FUNCTION_BLOCK FB_Tracking
VAR_IN_OUT
	stAxis  : ARRAY [GVL.cXP .. GVL.cXM] OF ST_AxisGroup;	
END_VAR
VAR_INPUT
	eCommand 			: E_Commands;
	bMotionDone			: BOOL;
	inReset				: ST_Reset;
	inMoveAxisAbsolute	: ST_MoveAxisAbsolute;
	inMoveAxisRelative	: ST_MoveAxisRelative;
END_VAR
VAR_OUTPUT
	stOutMotionDone : ST_MotionDone;
END_VAR
VAR
	//used in tracking Action
	stTrack			: ARRAY [0 .. 4] OF ST_TRACK;
	stTrackTemp		: ST_TRACK;
	bGoNextSeq		: BOOL;
	nAxisID			: INT;
	tTimeEnd		: T_DCTIME64;
	nMask			: ULINT := 16#FFFF_FFFF_0000_0000;
	
	//used in determining target duration
	fSpeed			: LREAL;
	tTargetDur		: LTIME;
	fDistance		: LREAL;
	
	fbMoving_Rtrig : ARRAY[0 .. 1] OF R_TRIG;
	fbRtrig		: ARRAY[GVL.cHallLower..GVL.cHallUpper] OF R_Trig;
	bInMotion	: BOOL;
	stMotionDone : ARRAY [0..1] OF ST_MotionDone;	
	nSequence	: DINT;
	nLastMoved	: INT;
	
	//counter
	i, j, k, m		: INT := 0;
	nTPC	: INT; //Trip Per Cycle
	
	//TestVar
	testRtrig : R_TRIG;
	testRtrig2 : R_TRIG;
	testInt: INT;
	testInt2: INT;
	testInt3: INT;
	testInt4: INT;
	testInt5: INT;
	testInt6: INT;
	testLREAL : LREAL;
	testTemp : ARRAY[0 .. 4] OF ST_Track;
	testTime : ARRAY[0 .. 4] OF T_DCTIME64;
	teststTrack : ARRAY[0 .. 4] OF T_DCTIME64;
	testDCTime	: ARRAY[0 .. 4] OF T_DCTIME64;
	nMask2	 : ULINT := 16#0000_0000_FFFF_FFFF;
	a, b : INT;
	
	
	
END_VAR

//////////////////////////////////////////////////////////////
//Algorithm for tracking blade position using hall switches	//
//////////////////////////////////////////////////////////////
stAxis[GVL.cXP].bTrackedFlag:=FALSE;
stAxis[GVL.cXM].bTrackedFlag:=FALSE;
nTPC:=0;
testInt3:=0;
testInt4:=0;

fbMoving_Rtrig[GVL.cXP](CLK:=stAxis[GVL.cXP].axisRef.Status.Moving);
IF fbMoving_Rtrig[GVL.cXP].Q THEN
	bInMotion:=TRUE;
	//AxisXP
	stMotionDone[GVL.cXP].axisNum := GVL.cXP;
	stMotionDone[GVL.cXP].nsamples := 0;
	stMotionDone[GVL.cXP].ntrans := 0;
	stMotionDone[gvl.cXP].startPos := stAxis[GVL.cXP].axisRef.NcToPlc.ActPos;
	stMotionDone[GVL.cXP].startTime := F_GetCurDcTaskTime64();
	stMotionDone[GVL.cXP].targetDur := LTIME#0D0H0M0S0MS0US0NS;
END_IF
fbMoving_Rtrig[GVL.cXM](CLK:=stAxis[GVL.cXM].axisRef.Status.Moving);
IF fbMoving_Rtrig[GVL.cXM].Q THEN
	bInMotion:=TRUE;
	//AxisXM
	stMotionDone[gvl.cXM].axisNum := GVL.cXM;
	stMotionDone[gvl.cXM].nsamples := 0;
	stMotionDone[gvl.cXM].ntrans := 0;
	stMotionDone[gvl.cXM].startPos := stAxis[GVL.cXM].axisRef.NcToPlc.ActPos;
	stMotionDone[gvl.cXM].startTime := F_GetCurDcTaskTime64();
	stMotionDone[gvl.cXM].targetDur := LTIME#0D0H0M0S0MS0US0NS;
END_IF

//determine target duration
IF eCommand = E_Commands.takeExposure THEN
	fSpeed	:= inReset.speed;
	IF (fSpeed>0) THEN
		IF (fSpeed>1668.355556) THEN
			fSpeed:=1668.355556;
		END_IF
		tTargetDur 	:= LREAL_TO_LTIME((2*GVL.cPosEnd)/(fSpeed)*EXPT(10,9));
	END_IF
ELSIF eCommand = E_Commands.moveAxisAbsolute THEN
	fDistance := ABS(stAxis[inMoveAxisAbsolute.axisIndex].axisRef.NcToPlc.ActPos - inMoveAxisAbsolute.position);
	fSpeed	:= inMoveAxisAbsolute.speed;
	IF (fSpeed>0) THEN
		IF (fSpeed>1668.355556) THEN
			fSpeed:=1668.355556;
		END_IF
		tTargetDur 	:= LREAL_TO_LTIME(((2*fDistance)/(fSpeed))*EXPT(10,9));
	END_IF
ELSIF eCommand = E_Commands.moveAxisRelative THEN
	tTargetDur	:= TIME_TO_LTIME(inMoveAxisRelative.moveTime);
END_IF

//Checks to see which blade set last moved
IF (stAxis[GVL.cXM].axisRef.Status.Moving AND stAxis[GVL.cXP].axisRef.Status.InTargetPosition) THEN
	nLastMoved:=GVL.cXM;
ELSIF (stAxis[GVL.cXP].axisRef.Status.Moving AND stAxis[GVL.cXM].axisRef.Status.InTargetPosition) THEN
	nLastMoved:=GVL.cXP;
END_IF
IF bMotionDone THEN
	//use for determining which blade set has finished during a travelling slit motion
	IF (stAxis[GVL.cXM].axisRef.Status.Moving AND stAxis[GVL.cXP].axisRef.Status.InTargetPosition) THEN
		nAxisID:=GVL.cXP;
	ELSIF (stAxis[GVL.cXP].axisRef.Status.Moving AND stAxis[GVL.cXM].axisRef.Status.InTargetPosition) THEN
		nAxisID:=GVL.cXM;
	ELSE 
		nAxisID:=nLastMoved;
	END_IF
	//bInMotion flag remains true if any of the blade set is still in motion
	IF ((NOT stAxis[GVL.cXP].axisRef.Status.Moving) AND (NOT stAxis[GVL.cXM].axisRef.Status.Moving)) THEN
		bInMotion := FALSE;
	END_IF
	nSequence := nSequence+1;
	tTimeEnd := F_GetCurDcTaskTime64();
	stMotionDone[nAxisID].actualDur := ULINT_TO_LTIME(tTimeEnd-stMotionDone[nAxisID].startTime);
	stMotionDone[nAxisID].targetDur := tTargetDur;
	stMotionDone[nAxisID].targetPos := stAxis[nAxisID].axisRef.NcToPlc.TargetPos;
	stMotionDone[nAxisID].endPos := stAxis[nAxisID].axisRef.NcToPlc.ActPos;
	
	stOutMotionDone:=stMotionDone[nAxisID];
	stOutMotionDone.sequence:=nSequence;
END_IF


//Detect hall switch transitions
FOR i:=GVL.cHallLower TO GVL.cHallUpper BY 1 DO
	fbRtrig[i](CLK:=GVL.nNumOfInputs[i].0);
	IF fbRtrig[i].Q THEN
		//identifies which hall switch tripped
		stTrack[nTPC].nSeqToCompare := INT_TO_WORD((i*10)+5);
		stTrack[nTPC].bEdgeToCompare := GVL.bInputEventState[i];
		stTrack[nTPC].nHallID := i;
		(*
			The time-stamping module only keeps track of the lower 32-bit time (about 4.29 seconds).
			To get the actual 64-bit time, add the acquired 32-bit time to the upper 32 bit of the DC time. 
			Check to see if the event time has overflowed by comparing appended time with current DC task time. 
			If appeneded time is greater than dc task time, then the 32-bit clock has overflowed.
			Decrement the 33rd bit of the appended time by 1 to get the correct time.
		*)
		stTrack[nTPC].tScanTime := (F_GetCurDcTaskTime64() AND nMask) + GVL.nInputEventTime[stTrack[nTPC].nHallID];
		IF stTrack[nTPC].tScanTime > F_GetCurDcTaskTime64() THEN
			stTrack[nTPC].tScanTIME := stTrack[nTPC].tScanTime - 16#1_0000_0000;
			testInt5:=testInt5+1;
		END_IF
		//increment the index
		nTPC:=nTPC+1;
		
		//Sort the data from lowest time to highest time
		IF nTPC>=2 THEN
			FOR j:=nTPC-1 TO 1 BY -1 DO
				IF (stTrack[j].tScanTime < stTrack[j-1].tScanTime) THEN
						stTrackTemp := stTrack[j];
						stTrack[j] := stTrack[j-1];
						stTrack[j-1] := stTrackTemp;
						testInt6 := testInt6+1;
				END_IF
			END_FOR
		END_IF

		
		//For debugging only: To see the highest number of trip per cycle
		testRTrig2(CLK:=(nTPC>=2));
		IF testRTrig2.Q THEN
			testInt3 := 1;
		END_IF
		testRTrig(CLK:=(nTPC>=3));
		IF testRTrig.Q THEN
			testTemp := stTrack;
			testInt4 := 1;
		END_IF
		IF m<nTPC THEN
			m:= nTPC;
		END_IF
		

			IF ((F_GetCurDcTaskTime64() - stTrack[0].tScanTime)>2000000) AND nTPC=1 THEN
				testTime[0]	:= F_GetCurDcTaskTime64() - stTrack[0].tScanTime;
				teststTrack[0] := stTrack[0].tScanTime;
				 testDCTime[0] := F_GetCurDcTaskTime64();
			END_IF
			IF ((F_GetCurDcTaskTime64() - stTrack[1].tScanTime)>2000000) AND nTPC=2 THEN
				testTime[1]	:= F_GetCurDcTaskTime64() - stTrack[1].tScanTime;
				teststTrack[1] := stTrack[1].tScanTime;
				testDCTime[1] := F_GetCurDcTaskTime64();
			END_IF
			IF ((F_GetCurDcTaskTime64() - stTrack[2].tScanTime)>2000000) AND nTPC=3 THEN
				testTime[2]	:= F_GetCurDcTaskTime64() - stTrack[2].tScanTime;
				teststTrack[2] := stTrack[2].tScanTime;
				testDCTime[2] := F_GetCurDcTaskTime64();
			END_IF
			IF ((F_GetCurDcTaskTime64() - stTrack[3].tScanTime)>2000000) AND nTPC=4 THEN
				testTime[3]	:= F_GetCurDcTaskTime64() - stTrack[3].tScanTime;
				teststTrack[3] := stTrack[3].tScanTime;
				testDCTime[3] := F_GetCurDcTaskTime64();
			END_IF
	END_IF
	
	//For debugging - checks to see if the same hall switch is tripped twice in one cycle
	IF GVL.nNumOfInputs[i]=2 THEN
		testInt:=testint+1;
	END_IF
	
END_FOR


	
//blade motion tracking
IF nTPC>0 THEN
	FOR k:=0 TO nTPC-1 BY 1 DO
		IF (stAxis[GVL.cXP].axisRef.Status.Moving AND stAxis[GVL.cXM].axisRef.Status.Moving) AND
			(stAxis[GVL.cXP].axisRef.Status.PositiveDirection AND stAxis[GVL.cXM].axisRef.Status.PositiveDirection) THEN
			ACT_TrackingDoublePositive();
		ELSIF (stAxis[GVL.cXP].axisRef.Status.Moving AND stAxis[GVL.cXM].axisRef.Status.Moving) AND
			(stAxis[GVL.cXP].axisRef.Status.NegativeDirection AND stAxis[GVL.cXM].axisRef.Status.NegativeDirection) THEN
			ACT_TrackingDoubleNegative();
		ELSE
			ACT_TrackingSingle();
		END_IF
		bGoNextSeq:=FALSE;
		IF nTPC=2 THEN
			testInt2:=testInt2+1;
		END_IF
	END_FOR
END_IF

ACTION ACT_TrackingDoubleNegative:
//Hall sensors position tracking for axis XP
IF stAxis[GVL.cXP].axisRef.Status.Moving THEN
	//Compare current sequence with recorded sequence. Update position if match. Negative direction.
	IF stAxis[GVL.cXP].axisRef.status.NegativeDirection AND stAxis[GVL.cXP].stHall[GVL.cDirNeg, stAxis[GVL.cXP].nTripCount].nSeq = stTrack[k].nSeqToCompare AND
			stAxis[GVL.cXP].stHall[GVL.cDirNeg, stAxis[GVL.cXP].nTripCount].bEdge = stTrack[k].bEdgeToCompare AND (NOT bGoNextSeq) THEN
		stAxis[GVL.cXP].fHallPosAct := stAxis[GVL.cXP].fHallPosCal[GVL.cDirNeg, stAxis[GVL.cXP].nTripCount];
		stAxis[GVL.cXP].nTripCount := stAxis[GVL.cXP].nTripCount - 1;		
		//track difference between hall sensor and encoder data at trip point
		stAxis[GVL.cXP].fPosDiffAtTrip := stAxis[GVL.cXP].axisRef.NcToPlc.ActPos - stAxis[GVL.cXP].fHallPosAct;
		stAxis[GVL.cXP].bTrackedFlag:=TRUE;
		bGoNextSeq:=TRUE;
		
		IF bInMotion AND MAIN.outShutterStatus.smState<>E_StatesMaint.Calibrating THEN
			nAxisID:= GVL.cXP;
			stMotionDone[GVL.cXP].trans[stMotionDone[GVL.cXP].ntrans].dcTime := stTrack[k].tScanTime;
			stMotionDone[GVL.cXP].trans[stMotionDone[GVL.cXP].ntrans].id := stTrack[k].nHallID;
			stMotionDone[GVL.cXP].trans[stMotionDone[GVL.cXP].ntrans].on := stTrack[k].bEdgeToCompare;
			stMotionDone[GVL.cXP].trans[stMotionDone[GVL.cXP].ntrans].pos := stAxis[GVL.cXP].fHallPosAct;
			stMotionDone[GVL.cXP].ntrans := stMotionDone[GVL.cXP].ntrans +1;
			
			stMotionDone[GVL.cXP].samples[stMotionDone[GVL.cXP].nsamples].dcTime := F_GetCurDcTaskTime64();
			stMotionDone[GVL.cXP].samples[stMotionDone[GVL.cXP].nsamples].pos := stAxis[GVL.cXP].axisRef.NcToPlc.ActPos;
			stMotionDone[GVL.cXP].nsamples := stMotionDone[GVL.cXP].nsamples + 1;
		END_IF
		
	END_IF
END_IF

//Hall sensors position tracking for axis XM
IF stAxis[GVL.cXM].axisRef.Status.Moving THEN
	//Compare current sequence with recorded sequence. Update position if match. Negative direction.
	IF stAxis[GVL.cXM].axisRef.status.NegativeDirection AND stAxis[GVL.cXM].stHall[GVL.cDirNeg, stAxis[GVL.cXM].nTripCount].nSeq = stTrack[k].nSeqToCompare AND
			stAxis[GVL.cXM].stHall[GVL.cDirNeg, stAxis[GVL.cXM].nTripCount].bEdge = stTrack[k].bEdgeToCompare AND (NOT bGoNextSeq) THEN
		stAxis[GVL.cXM].fHallPosAct := stAxis[GVL.cXM].fHallPosCal[GVL.cDirNeg, stAxis[GVL.cXM].nTripCount];
		stAxis[GVL.cXM].nTripCount := stAxis[GVL.cXM].nTripCount + 1;	
		//track difference between hall sensor and encoder data at trip point
		stAxis[GVL.cXM].fPosDiffAtTrip := stAxis[GVL.cXM].axisRef.NcToPlc.ActPos - stAxis[GVL.cXM].fHallPosAct;
		stAxis[GVL.cXM].bTrackedFlag:=TRUE;
		bGoNextSeq:=TRUE;
		
		IF bInMotion AND MAIN.outShutterStatus.smState<>E_StatesMaint.Calibrating THEN
			nAxisID:= GVL.cXM;
			stMotionDone[GVL.cXM].trans[stMotionDone[GVL.cXM].ntrans].dcTime := stTrack[k].tScanTime;
			stMotionDone[GVL.cXM].trans[stMotionDone[GVL.cXM].ntrans].id := stTrack[k].nHallID;
			stMotionDone[GVL.cXM].trans[stMotionDone[GVL.cXM].ntrans].on := stTrack[k].bEdgeToCompare;
			stMotionDone[GVL.cXM].trans[stMotionDone[GVL.cXM].ntrans].pos := stAxis[GVL.cXM].fHallPosAct;
			stMotionDone[GVL.cXM].ntrans := stMotionDone[GVL.cXM].ntrans +1;
			
			stMotionDone[GVL.cXM].samples[stMotionDone[GVL.cXM].nsamples].dcTime := F_GetCurDcTaskTime64();
			stMotionDone[GVL.cXM].samples[stMotionDone[GVL.cXM].nsamples].pos := stAxis[GVL.cXM].axisRef.NcToPlc.ActPos;
			stMotionDone[GVL.cXM].nsamples := stMotionDone[GVL.cXM].nsamples + 1;
		END_IF
		
	END_IF
END_IF
END_ACTION

ACTION ACT_TrackingDoublePositive:
//Hall sensors position tracking for axis XM
IF stAxis[GVL.cXM].axisRef.Status.Moving THEN
	//Compare current sequence with recorded sequence. Update position if match. Positive direction.
	IF stAxis[GVL.cXM].axisRef.status.PositiveDirection AND stAxis[GVL.cXM].stHall[GVL.cDirPos, stAxis[GVL.cXM].nTripCount].nSeq = stTrack[k].nSeqToCompare AND
			stAxis[GVL.cXM].stHall[GVL.cDirPos, stAxis[GVL.cXM].nTripCount].bEdge = stTrack[k].bEdgeToCompare AND (NOT bGoNextSeq) THEN
		stAxis[GVL.cXM].fHallPosAct := stAxis[GVL.cXM].fHallPosCal[GVL.cDirPos, stAxis[GVL.cXM].nTripCount];
		stAxis[GVL.cXM].nTripCount := stAxis[GVL.cXM].nTripCount - 1;	
		//track difference between hall sensor and encoder data at trip point
		stAxis[GVL.cXM].fPosDiffAtTrip := stAxis[GVL.cXM].axisRef.NcToPlc.ActPos - stAxis[GVL.cXM].fHallPosAct;
		stAxis[GVL.cXM].bTrackedFlag:=TRUE;
		bGoNextSeq:=TRUE;
		
		IF bInMotion AND MAIN.outShutterStatus.smState<>E_StatesMaint.Calibrating THEN
			nAxisID:= GVL.cXM;
			stMotionDone[GVL.cXM].trans[stMotionDone[GVL.cXM].ntrans].dcTime := stTrack[k].tScanTime;
			stMotionDone[GVL.cXM].trans[stMotionDone[GVL.cXM].ntrans].id := stTrack[k].nHallID;
			stMotionDone[GVL.cXM].trans[stMotionDone[GVL.cXM].ntrans].on := stTrack[k].bEdgeToCompare;
			stMotionDone[GVL.cXM].trans[stMotionDone[GVL.cXM].ntrans].pos := stAxis[GVL.cXM].fHallPosAct;
			stMotionDone[GVL.cXM].ntrans := stMotionDone[GVL.cXM].ntrans +1;
			
			stMotionDone[GVL.cXM].samples[stMotionDone[GVL.cXM].nsamples].dcTime := F_GetCurDcTaskTime64();
			stMotionDone[GVL.cXM].samples[stMotionDone[GVL.cXM].nsamples].pos := stAxis[GVL.cXM].axisRef.NcToPlc.ActPos;
			stMotionDone[GVL.cXM].nsamples := stMotionDone[GVL.cXM].nsamples + 1;
		END_IF
		
	END_IF
END_IF

//Hall sensors position tracking for axis XP
IF stAxis[GVL.cXP].axisRef.Status.Moving THEN
	//Compare current sequence with recorded sequence. Update position if match. Positive direction.
	IF stAxis[GVL.cXP].axisRef.status.PositiveDirection AND stAxis[GVL.cXP].stHall[GVL.cDirPos, stAxis[GVL.cXP].nTripCount].nSeq = stTrack[k].nSeqToCompare AND 
			stAxis[GVL.cXP].stHall[GVL.cDirPos, stAxis[GVL.cXP].nTripCount].bEdge = stTrack[k].bEdgeToCompare AND (NOT bGoNextSeq) THEN
		stAxis[GVL.cXP].fHallPosAct := stAxis[GVL.cXP].fHallPosCal[GVL.cDirPos, stAxis[GVL.cXP].nTripCount];
		stAxis[GVL.cXP].nTripCount := stAxis[GVL.cXP].nTripCount + 1;
		//track difference between hall sensor and encoder data at trip point
		stAxis[GVL.cXP].fPosDiffAtTrip := stAxis[GVL.cXP].axisRef.NcToPlc.ActPos - stAxis[GVL.cXP].fHallPosAct;
		stAxis[GVL.cXP].bTrackedFlag:=TRUE;
		bGoNextSeq:=TRUE;
		
		IF bInMotion AND MAIN.outShutterStatus.smState<>E_StatesMaint.Calibrating THEN
			nAxisID:= GVL.cXP;
			stMotionDone[GVL.cXP].trans[stMotionDone[GVL.cXP].ntrans].dcTime := stTrack[k].tScanTime;
			stMotionDone[GVL.cXP].trans[stMotionDone[GVL.cXP].ntrans].id := stTrack[k].nHallID;
			stMotionDone[GVL.cXP].trans[stMotionDone[GVL.cXP].ntrans].on := stTrack[k].bEdgeToCompare;
			stMotionDone[GVL.cXP].trans[stMotionDone[GVL.cXP].ntrans].pos := stAxis[GVL.cXP].fHallPosAct;
			stMotionDone[GVL.cXP].ntrans := stMotionDone[GVL.cXP].ntrans +1;
			
			stMotionDone[GVL.cXP].samples[stMotionDone[GVL.cXP].nsamples].dcTime := F_GetCurDcTaskTime64();
			stMotionDone[GVL.cXP].samples[stMotionDone[GVL.cXP].nsamples].pos := stAxis[GVL.cXP].axisRef.NcToPlc.ActPos;
			stMotionDone[GVL.cXP].nsamples := stMotionDone[GVL.cXP].nsamples + 1;
		END_IF
		
	END_IF
END_IF
END_ACTION

ACTION ACT_TrackingSingle:
//Hall sensors position tracking for axis XP
IF stAxis[GVL.cXP].axisRef.Status.Moving THEN
	//Compare current sequence with recorded sequence. Update position if match. Positive direction.
	IF stAxis[GVL.cXP].axisRef.status.PositiveDirection AND stAxis[GVL.cXP].stHall[GVL.cDirPos, stAxis[GVL.cXP].nTripCount].nSeq = stTrack[k].nSeqToCompare AND 
			stAxis[GVL.cXP].stHall[GVL.cDirPos, stAxis[GVL.cXP].nTripCount].bEdge = stTrack[k].bEdgeToCompare AND (NOT bGoNextSeq) THEN
		stAxis[GVL.cXP].fHallPosAct := stAxis[GVL.cXP].fHallPosCal[GVL.cDirPos, stAxis[GVL.cXP].nTripCount];
		stAxis[GVL.cXP].nTripCount := stAxis[GVL.cXP].nTripCount + 1;
		//track difference between hall sensor and encoder data at trip point
		stAxis[GVL.cXP].fPosDiffAtTrip := stAxis[GVL.cXP].axisRef.NcToPlc.ActPos - stAxis[GVL.cXP].fHallPosAct;
		stAxis[GVL.cXP].bTrackedFlag:=TRUE;
		bGoNextSeq:=TRUE;
		
		IF bInMotion AND MAIN.outShutterStatus.smState<>E_StatesMaint.Calibrating THEN
			nAxisID:= GVL.cXP;
			stMotionDone[GVL.cXP].trans[stMotionDone[GVL.cXP].ntrans].dcTime := stTrack[k].tScanTime;
			stMotionDone[GVL.cXP].trans[stMotionDone[GVL.cXP].ntrans].id := stTrack[k].nHallID;
			stMotionDone[GVL.cXP].trans[stMotionDone[GVL.cXP].ntrans].on := stTrack[k].bEdgeToCompare;
			stMotionDone[GVL.cXP].trans[stMotionDone[GVL.cXP].ntrans].pos := stAxis[GVL.cXP].fHallPosAct;
			stMotionDone[GVL.cXP].ntrans := stMotionDone[GVL.cXP].ntrans +1;
			
			stMotionDone[GVL.cXP].samples[stMotionDone[GVL.cXP].nsamples].dcTime := F_GetCurDcTaskTime64();
			stMotionDone[GVL.cXP].samples[stMotionDone[GVL.cXP].nsamples].pos := stAxis[GVL.cXP].axisRef.NcToPlc.ActPos;
			stMotionDone[GVL.cXP].nsamples := stMotionDone[GVL.cXP].nsamples + 1;
		END_IF
		
	END_IF
	//Compare current sequence with recorded sequence. Update position if match. Negative direction.
	IF stAxis[GVL.cXP].axisRef.status.NegativeDirection AND stAxis[GVL.cXP].stHall[GVL.cDirNeg, stAxis[GVL.cXP].nTripCount].nSeq = stTrack[k].nSeqToCompare AND
			stAxis[GVL.cXP].stHall[GVL.cDirNeg, stAxis[GVL.cXP].nTripCount].bEdge = stTrack[k].bEdgeToCompare AND (NOT bGoNextSeq) THEN
		stAxis[GVL.cXP].fHallPosAct := stAxis[GVL.cXP].fHallPosCal[GVL.cDirNeg, stAxis[GVL.cXP].nTripCount];
		stAxis[GVL.cXP].nTripCount := stAxis[GVL.cXP].nTripCount - 1;		
		//track difference between hall sensor and encoder data at trip point
		stAxis[GVL.cXP].fPosDiffAtTrip := stAxis[GVL.cXP].axisRef.NcToPlc.ActPos - stAxis[GVL.cXP].fHallPosAct;
		stAxis[GVL.cXP].bTrackedFlag:=TRUE;
		bGoNextSeq:=TRUE;
		
		IF bInMotion AND MAIN.outShutterStatus.smState<>E_StatesMaint.Calibrating THEN
			nAxisID:= GVL.cXP;
			stMotionDone[GVL.cXP].trans[stMotionDone[GVL.cXP].ntrans].dcTime := stTrack[k].tScanTime;
			stMotionDone[GVL.cXP].trans[stMotionDone[GVL.cXP].ntrans].id := stTrack[k].nHallID;
			stMotionDone[GVL.cXP].trans[stMotionDone[GVL.cXP].ntrans].on := stTrack[k].bEdgeToCompare;
			stMotionDone[GVL.cXP].trans[stMotionDone[GVL.cXP].ntrans].pos := stAxis[GVL.cXP].fHallPosAct;
			stMotionDone[GVL.cXP].ntrans := stMotionDone[GVL.cXP].ntrans +1;
			
			stMotionDone[GVL.cXP].samples[stMotionDone[GVL.cXP].nsamples].dcTime := F_GetCurDcTaskTime64();
			stMotionDone[GVL.cXP].samples[stMotionDone[GVL.cXP].nsamples].pos := stAxis[GVL.cXP].axisRef.NcToPlc.ActPos;
			stMotionDone[GVL.cXP].nsamples := stMotionDone[GVL.cXP].nsamples + 1;
		END_IF
		
	END_IF
END_IF

//Hall sensors position tracking for axis XM
IF stAxis[GVL.cXM].axisRef.Status.Moving THEN
	//Compare current sequence with recorded sequence. Update position if match. Positive direction.
	IF stAxis[GVL.cXM].axisRef.status.PositiveDirection AND stAxis[GVL.cXM].stHall[GVL.cDirPos, stAxis[GVL.cXM].nTripCount].nSeq = stTrack[k].nSeqToCompare AND
			stAxis[GVL.cXM].stHall[GVL.cDirPos, stAxis[GVL.cXM].nTripCount].bEdge = stTrack[k].bEdgeToCompare AND (NOT bGoNextSeq) THEN
		stAxis[GVL.cXM].fHallPosAct := stAxis[GVL.cXM].fHallPosCal[GVL.cDirPos, stAxis[GVL.cXM].nTripCount];
		stAxis[GVL.cXM].nTripCount := stAxis[GVL.cXM].nTripCount - 1;	
		//track difference between hall sensor and encoder data at trip point
		stAxis[GVL.cXM].fPosDiffAtTrip := stAxis[GVL.cXM].axisRef.NcToPlc.ActPos - stAxis[GVL.cXM].fHallPosAct;
		stAxis[GVL.cXM].bTrackedFlag:=TRUE;
		bGoNextSeq:=TRUE;
		
		IF bInMotion AND MAIN.outShutterStatus.smState<>E_StatesMaint.Calibrating THEN
			nAxisID:= GVL.cXM;
			stMotionDone[GVL.cXM].trans[stMotionDone[GVL.cXM].ntrans].dcTime := stTrack[k].tScanTime;
			stMotionDone[GVL.cXM].trans[stMotionDone[GVL.cXM].ntrans].id := stTrack[k].nHallID;
			stMotionDone[GVL.cXM].trans[stMotionDone[GVL.cXM].ntrans].on := stTrack[k].bEdgeToCompare;
			stMotionDone[GVL.cXM].trans[stMotionDone[GVL.cXM].ntrans].pos := stAxis[GVL.cXM].fHallPosAct;
			stMotionDone[GVL.cXM].ntrans := stMotionDone[GVL.cXM].ntrans +1;
			
			stMotionDone[GVL.cXM].samples[stMotionDone[GVL.cXM].nsamples].dcTime := F_GetCurDcTaskTime64();
			stMotionDone[GVL.cXM].samples[stMotionDone[GVL.cXM].nsamples].pos := stAxis[GVL.cXM].axisRef.NcToPlc.ActPos;
			stMotionDone[GVL.cXM].nsamples := stMotionDone[GVL.cXM].nsamples + 1;
		END_IF
		
	END_IF
	//Compare current sequence with recorded sequence. Update position if match. Negative direction.
	IF stAxis[GVL.cXM].axisRef.status.NegativeDirection AND stAxis[GVL.cXM].stHall[GVL.cDirNeg, stAxis[GVL.cXM].nTripCount].nSeq = stTrack[k].nSeqToCompare AND
			stAxis[GVL.cXM].stHall[GVL.cDirNeg, stAxis[GVL.cXM].nTripCount].bEdge = stTrack[k].bEdgeToCompare AND (NOT bGoNextSeq) THEN
		stAxis[GVL.cXM].fHallPosAct := stAxis[GVL.cXM].fHallPosCal[GVL.cDirNeg, stAxis[GVL.cXM].nTripCount];
		stAxis[GVL.cXM].nTripCount := stAxis[GVL.cXM].nTripCount + 1;	
		//track difference between hall sensor and encoder data at trip point
		stAxis[GVL.cXM].fPosDiffAtTrip := stAxis[GVL.cXM].axisRef.NcToPlc.ActPos - stAxis[GVL.cXM].fHallPosAct;
		stAxis[GVL.cXM].bTrackedFlag:=TRUE;
		bGoNextSeq:=TRUE;
		
		IF bInMotion AND MAIN.outShutterStatus.smState<>E_StatesMaint.Calibrating THEN
			nAxisID:= GVL.cXM;
			stMotionDone[GVL.cXM].trans[stMotionDone[GVL.cXM].ntrans].dcTime := stTrack[k].tScanTime;
			stMotionDone[GVL.cXM].trans[stMotionDone[GVL.cXM].ntrans].id := stTrack[k].nHallID;
			stMotionDone[GVL.cXM].trans[stMotionDone[GVL.cXM].ntrans].on := stTrack[k].bEdgeToCompare;
			stMotionDone[GVL.cXM].trans[stMotionDone[GVL.cXM].ntrans].pos := stAxis[GVL.cXM].fHallPosAct;
			stMotionDone[GVL.cXM].ntrans := stMotionDone[GVL.cXM].ntrans +1;
			
			stMotionDone[GVL.cXM].samples[stMotionDone[GVL.cXM].nsamples].dcTime := F_GetCurDcTaskTime64();
			stMotionDone[GVL.cXM].samples[stMotionDone[GVL.cXM].nsamples].pos := stAxis[GVL.cXM].axisRef.NcToPlc.ActPos;
			stMotionDone[GVL.cXM].nsamples := stMotionDone[GVL.cXM].nsamples + 1;
		END_IF
		
	END_IF
END_IF
END_ACTION

END_FUNCTION_BLOCK

(* stored: Version 1.1.0.1, ProductVersion 3.1.4020.12
   POU FB_Tracking: Id {462a5933-fe60-42d4-a574-27170521c4c5}, SpecialFunc None
   Action ACT_TrackingDoubleNegative: Id {0039cb21-b703-43f6-867c-8fbe57c73e86}
   Action ACT_TrackingDoublePositive: Id {015fe346-39d0-42ba-a488-79403589a261}
   Action ACT_TrackingSingle: Id {68bb727f-4301-4350-9f19-54a85b8d6b0c} *)
